FUNCTION_BLOCK EL2809
VAR
	{attribute addProperty Name "CHANNEL_"}
	_io : EL2809_Data;
	{attribute addProperty Name "Info data"}
	_infoData : InfoDataBase;
	{attribute addProperty Name "WcState"}
	_wcState : WcStateBase;
END_VAR

_infoData();

PROPERTY IO : REFERENCE TO EL2809_Data
GET
IO REF= _io;
END_GET
END_PROPERTY

END_FUNCTION_BLOCK

(* stored: Version 1.1.0.1, ProductVersion 3.1.4024.9
   POU EL2809: Id {a5d8806d-2fa9-0a34-239c-97db45246e10}, SpecialFunc None
   Property IO: Id {85b3b5a7-679e-0afe-1f4f-a394a1bac951}
   Get Get: Id {02ea8413-b717-0fcd-2401-f6ab7af0ed4d} *)
